{attribute 'qualified_only'}
{attribute 'strict'}
TYPE E_Pixii_VendorSpecificStatusCode :
(
	eNoError := 0,
	eModbusTCPError := 1,
	ePixiiError := 2
);
END_TYPE

(* stored: Version 1.1.0.1, ProductVersion 3.1.4024.12
   DUT E_Pixii_VendorSpecificStatusCode: Id {73a3e2a7-f4d5-46a7-872a-0b4bca2c2b23} *)
